Staubli VAL3: sad_project_1.dtx

public num Ref_Vel
public mdesc mNomSpeed = {tmax=100, rmax=100, leave=0.1, reach=0.1, blend=off}
public jointRx Jnt_cnfg = {j3=90, j5=90, j6=90}
public tool tTool = {z=200, fatherId=flange[0], ioLink=valve1}
public frame fReference = {x=1365.054, y=-125.975, z=-500, fatherId=world[0]}
public pointRx Pnt_1st_lyr[2]
  [0] = {y=-1000, rx=-180, rz=-90, shoulder=lefty, elbow=epositive, wrist=wpositive, fatherId=fReference[0]}
  [1] = {y=1000, rx=-180, rz=-90, shoulder=lefty, elbow=epositive, wrist=wpositive, fatherId=fReference[0]}
public pointRx Pnt_2nd_lyr[4]
  [0] = {y=1000, z=77, rx=180, rz=-90, shoulder=lefty, elbow=epositive, wrist=wpositive, fatherId=fReference[0]}
  [1] = {y=-1000, z=77, rx=180, rz=-90, shoulder=lefty, elbow=epositive, wrist=wpositive, fatherId=fReference[0]}
  [2] = {y=-1000, z=22, rx=180, rz=-90, shoulder=lefty, elbow=epositive, wrist=wpositive, fatherId=fReference[0]}
  [3] = {y=1000, z=22, rx=180, rz=-90, shoulder=lefty, elbow=epositive, wrist=wpositive, fatherId=fReference[0]}
public pointRx Pnt_3rd_lyr[4]
  [0] = {y=1000, z=99, rx=180, rz=-90, shoulder=lefty, elbow=epositive, wrist=wpositive, fatherId=fReference[0]}
  [1] = {y=-1000, z=99, rx=180, rz=-90, shoulder=lefty, elbow=epositive, wrist=wpositive, fatherId=fReference[0]}
  [2] = {y=-1000, z=44, rx=180, rz=-90, shoulder=lefty, elbow=epositive, wrist=wpositive, fatherId=fReference[0]}
  [3] = {y=1000, z=44, rx=180, rz=-90, shoulder=lefty, elbow=epositive, wrist=wpositive, fatherId=fReference[0]}
public pointRx Pnt_4th_lyr[4]
  [0] = {y=1000, z=116, rx=180, rz=-90, shoulder=lefty, elbow=epositive, wrist=wpositive, fatherId=fReference[0]}
  [1] = {y=-1000, z=116, rx=180, rz=-90, shoulder=lefty, elbow=epositive, wrist=wpositive, fatherId=fReference[0]}
  [2] = {y=-1000, z=66, rx=180, rz=-90, shoulder=lefty, elbow=epositive, wrist=wpositive, fatherId=fReference[0]}
  [3] = {y=1000, z=66, rx=180, rz=-90, shoulder=lefty, elbow=epositive, wrist=wpositive, fatherId=fReference[0]}
public trsf trTrsf
sio sioASCII = {link=Socket\trsf_sv}
public bool check_status
public bool spd_cntl
public mdesc cnst_vel = {tmax=100, rmax=100, leave=0.1, reach=0.1, blend=cartesian}
aio Tpompe
dio doValve1
dio doValve2
